// TIA Portal V17 export
// export: Created 2024-08-09T12:53:02.6201975Z, ExportSetting WithDefaults, DisplayName Totally Integrated Automation Portal, DisplayVersion V17 Update 7, DisplayName TIA Portal Openness, DisplayVersion V17 Update 7, DisplayName TIA Portal Version Control Interface, DisplayVersion V17, DisplayName STEP 7 Professional, DisplayVersion V17 Update 7, DisplayName STEP 7 Safety, DisplayVersion V17 Update 6, DisplayName WinCC Professional, DisplayVersion V17 Update 7
DATA_BLOCK "Test_Dosage_DB"   // DB11
VERSION : 0.1
// stored: AutoNumber true, DBAccessibleFromOPCUA true, DBAccessibleFromWebserver true, InstanceOfName Test_Dosage, InstanceOfType FB
"Test_Dosage"
   // VAR
   //    "Pt_Zs(LotS1S2BP1)" { S7_SetPoint := 'True'} : "S_Suivi_Dosage";
   //    Zone_Suivi : SInt;
   //    LotS1S2BP1 : Bool;
   //    CIRCUIT : "S_Circuit";
   //    RAZ_Pt_Zs { ExternalAccessible := 'False'; ExternalVisible := 'False'; ExternalWritable := 'False'} : "S_Suivi_Dosage";
   // END_VAR
BEGIN
END_DATA_BLOCK
